Fanuc KAREL source: ka00077.KL

PROGRAM KA00077
%STACKSIZE=65535
%PRIORITY=65535
%NOLOCKGROUP
VAR
SRC : XYZWPREXT
DST : POSITION
BEGIN
SRC.X=1.0
-- UNSAFE_SOURCE_IR line 8: DST = convert_xyzwprext_to_position(SRC)
END KA00077
